{attribute 'GeneratedUsingTerminal: CU1124-0000-0016'}
{attribute addProperty BoxType "CU1124-0000-0016"}
{attribute addProperty Id "A_0004_CU1128_0000_0000A_0004_CU1128_0000_0000_A9D31A95124"}
{attribute addProperty CRC "3519238464"}
{attribute addProperty Size "124"}
TYPE A_0003_CU1124_0000_0016_D1C35140 EXTENDS CU1124_AB5A9467 :
STRUCT
	{attribute addProperty Name "A_0004_CU1128_0000_0000"}
	{attribute addProperty PreviousPort "A_0003(CU1124-0000-0016) : D"}
	A_0004_CU1128_0000_0000 : A_0004_CU1128_0000_0000_A9D31A95;
END_STRUCT
END_TYPE

(* stored: Version 1.2.0.0, ProductVersion 3.1.4024.9
   DUT A_0003_CU1124_0000_0016_D1C35140: Id {0fbd0f81-7ed7-4b1e-b8d5-46f77d8604dc} *)
